// TIA Portal V18 export
// export: Created 2026-06-11T11:10:30.5736779Z, ExportSetting WithDefaults, DisplayName Totally Integrated Automation Portal, DisplayVersion V18, DisplayName TIA Portal Openness, DisplayVersion V18, DisplayName TIA Portal Version Control Interface, DisplayVersion V18, DisplayName STEP 7 Professional, DisplayVersion V18, DisplayName STEP 7 Safety, DisplayVersion V18, DisplayName WinCC Professional, DisplayVersion V18
VAR_GLOBAL   // PLC tag table "PLC_Simulation_Tags"
   "1400_FT115_PV" AT %MD100 : Real;   // Lưu lượng dòng liệu đo được tại FT115
   "1400_FT101_PV" AT %MD104 : Real;   // Lưu lượng dòng liệu đo được tại FT101
   "1400_1_02_PV" AT %MD108 : Real;   // Giá trị đo của cảm biến 1-02
   "1406_TX35_PV" AT %MD112 : Real;   // Giá trị đo cảm biến nhiệt độ/áp suất TX35
   "1400_TT64_PV" AT %MD116 : Real;   // Nhiệt độ đo được tại TT64
   "1400_TT32_PV" AT %MD120 : Real;   // Nhiệt độ đo được tại TT32
   "1400_LGFE01_PV" AT %MD124 : Real;   // Mức bồn hoặc lưu lượng đo tại LGFE01
   "1400_FS51_PV" AT %MD128 : Real;   // Giá trị lưu lượng đo được tại FS51
   "1400_FY301_PV" AT %MD132 : Real;   // Mức cân hoặc vị trí điều khiển bồn FY301
   "1400_TT101_PV" AT %MD136 : Real;   // Nhiệt độ đo được tại TT101
   "1400_FTT02_PV" AT %MD140 : Real;   // Lưu lượng/nhiệt độ đo được tại FTT02
   "1500S_Trang_Thai" AT %M200.0 : Bool;   // Trạng thái hoạt động dòng liệu 1500S (0: Không chảy, 1: Đang chảy)
   "1404T_Trang_Thai" AT %M200.1 : Bool;   // Trạng thái hoạt động dòng liệu 1404T
   CR_2013_FO_104_Trang_Thai AT %M200.2 : Bool;   // Trạng thái hoạt động dòng liệu CR-2013-FO-104
   BFOC_SS_20_06_Trang_Thai AT %M200.3 : Bool;   // Trạng thái hoạt động dòng liệu BFOC-SS-20-06
   PC03010T01_Trang_Thai AT %M200.4 : Bool;   // Trạng thái dòng liệu đầu ra PC03010T01
   "1401_Trang_Thai" AT %M200.5 : Bool;   // Trạng thái dòng liệu xả đáy 1401
   "1400_PT91_Chay" AT %M200.6 : Bool;   // Tín hiệu báo chạy bơm 1400PT91 (1: Chạy)
   "1400_KCK01_Chay" AT %M200.7 : Bool;   // Tín hiệu báo chạy cánh khuấy bồn 1400KCK01
   "1400_FT102_Mo" AT %M201.0 : Bool;   // Tín hiệu báo mở van nạp liệu 1400FT102
   "1400_TY33_Mo" AT %M201.1 : Bool;   // Tín hiệu báo mở van điều khiển cooling 1400TY33
   "160_FEC53_Mo" AT %M201.2 : Bool;   // Tín hiệu báo mở van kẹp 160 FEC53
   "1400_TXC32_Mo" AT %M201.3 : Bool;   // Tín hiệu báo mở van điều khiển 1400TXC32
   "1400_TC32_Mo" AT %M201.4 : Bool;   // Tín hiệu báo mở van điều khiển 1400TC32
   "1400_FIC01_Mo" AT %M201.5 : Bool;   // Tín hiệu báo mở van điều khiển 1400FIC01
   "1400_FS51_Mo" AT %M201.6 : Bool;   // Tín hiệu báo mở van xả đáy 1400FS51
   "1500S_Status" AT %MW300 : Int;   // Mã trạng thái dòng liệu 1500S (0: Dừng, 1: Chạy, 2: Lỗi)
   "1404T_Status" AT %MW302 : Int;   // Mã trạng thái dòng liệu 1404T
   CR_2013_FO_104_Status AT %MW304 : Int;   // Mã trạng thái dòng liệu CR-2013-FO-104
   BFOC_SS_20_06_Status AT %MW306 : Int;   // Mã trạng thái dòng liệu BFOC-SS-20-06
   PC03010T01_Status AT %MW308 : Int;   // Mã trạng thái dòng liệu PC03010T01
   "1401_Status" AT %MW310 : Int;   // Mã trạng thái dòng liệu xả đáy 1401
   "1400_PT91_Status" AT %MW312 : Int;   // Mã trạng thái hoạt động bơm 1400PT91 (0: Dừng, 1: Chạy, 2: Lỗi)
   "1400_KCK01_Status" AT %MW314 : Int;   // Mã trạng thái hoạt động cánh khuấy 1400KCK01
   "1400_FT102_Status" AT %MW316 : Int;   // Mã trạng thái hoạt động van 1400FT102 (0: Đóng, 1: Mở, 2: Lỗi)
   "1400_TY33_Status" AT %MW318 : Int;   // Mã trạng thái hoạt động van 1400TY33
   "160_FEC53_Status" AT %MW320 : Int;   // Mã trạng thái hoạt động van 160 FEC53
   "1400_TXC32_Status" AT %MW322 : Int;   // Mã trạng thái hoạt động van 1400TXC32
   "1400_TC32_Status" AT %MW324 : Int;   // Mã trạng thái hoạt động van 1400TC32
   "1400_FIC01_Status" AT %MW326 : Int;   // Mã trạng thái hoạt động van 1400FIC01
   "1400_FS51_Status" AT %MW328 : Int;   // Mã trạng thái hoạt động van 1400FS51
   Sim_Counter AT %MD400 : Real;   // Biến đếm trung gian cho sóng tam giác mô phỏng
   Sim_Dir AT %M404.0 : Bool;   // Bit hướng đếm mô phỏng (0: Tăng, 1: Giảm)
   Sim_Val_Norm AT %MD408 : Real;   // Giá trị đếm đã chuẩn hóa về dải 0.0 - 1.0
   Timer_Sim_Pulse_Output AT %M404.1 : Bool;   // Xung kích hoạt đếm từ Timer
END_VAR
